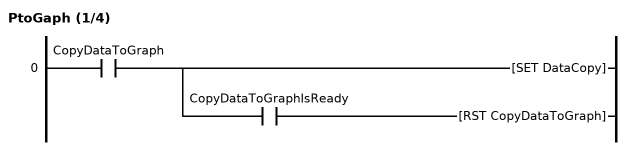
[picture p24: ladder of PtoGaph, rungs at steps 0 to 0]
0     LD      CopyDataToGraph
      SET     DataCopy
      AND     CopyDataToGraphIsReady
      RST     CopyDataToGraph
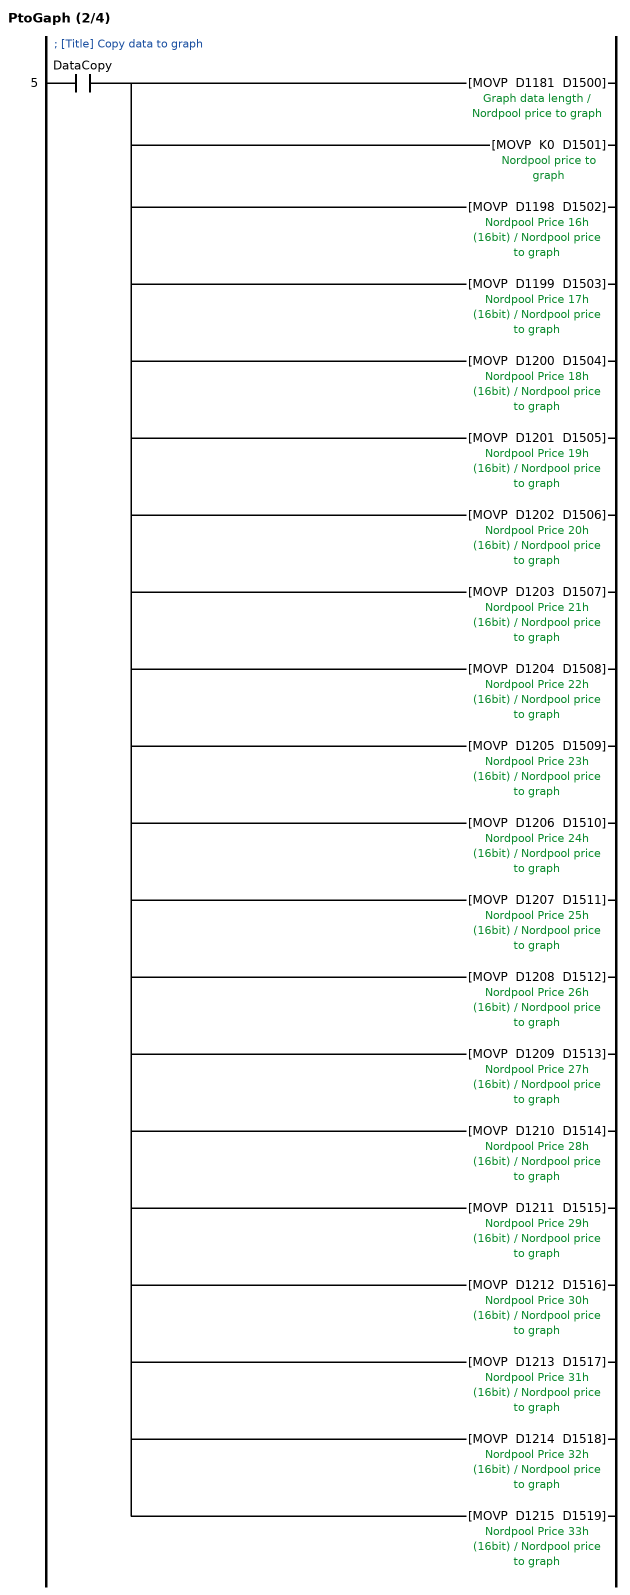
; [Title] Copy data to graph
5     LD      DataCopy
      MOVP    D1181 D1500  ; Graph data length / Nordpool price to graph
      MOVP    K0 D1501  ; Nordpool price to graph
      MOVP    D1198 D1502  ; Nordpool Price 16h (16bit) / Nordpool price to graph
      MOVP    D1199 D1503  ; Nordpool Price 17h (16bit) / Nordpool price to graph
      MOVP    D1200 D1504  ; Nordpool Price 18h (16bit) / Nordpool price to graph
      MOVP    D1201 D1505  ; Nordpool Price 19h (16bit) / Nordpool price to graph
      MOVP    D1202 D1506  ; Nordpool Price 20h (16bit) / Nordpool price to graph
      MOVP    D1203 D1507  ; Nordpool Price 21h (16bit) / Nordpool price to graph
      MOVP    D1204 D1508  ; Nordpool Price 22h (16bit) / Nordpool price to graph
      MOVP    D1205 D1509  ; Nordpool Price 23h (16bit) / Nordpool price to graph
      MOVP    D1206 D1510  ; Nordpool Price 24h (16bit) / Nordpool price to graph
      MOVP    D1207 D1511  ; Nordpool Price 25h (16bit) / Nordpool price to graph
      MOVP    D1208 D1512  ; Nordpool Price 26h (16bit) / Nordpool price to graph
      MOVP    D1209 D1513  ; Nordpool Price 27h (16bit) / Nordpool price to graph
      MOVP    D1210 D1514  ; Nordpool Price 28h (16bit) / Nordpool price to graph
      MOVP    D1211 D1515  ; Nordpool Price 29h (16bit) / Nordpool price to graph
      MOVP    D1212 D1516  ; Nordpool Price 30h (16bit) / Nordpool price to graph
      MOVP    D1213 D1517  ; Nordpool Price 31h (16bit) / Nordpool price to graph
      MOVP    D1214 D1518  ; Nordpool Price 32h (16bit) / Nordpool price to graph
      MOVP    D1215 D1519  ; Nordpool Price 33h (16bit) / Nordpool price to graph
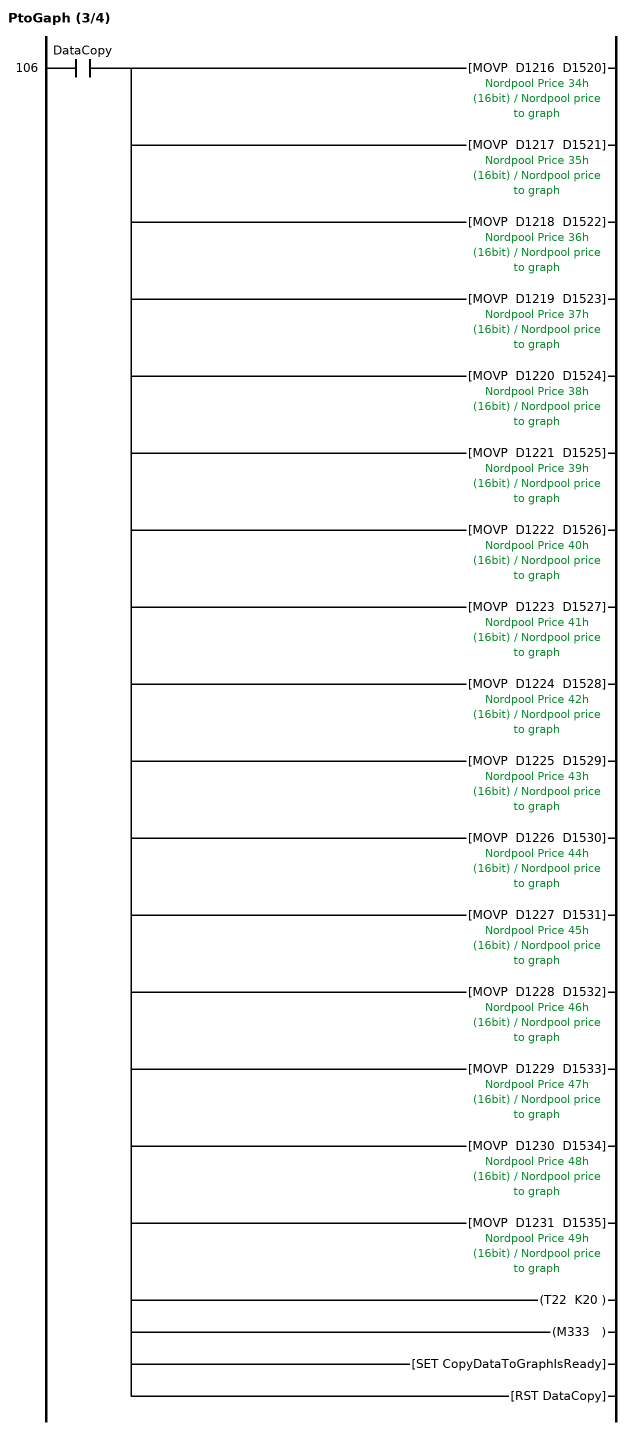
106   LD      DataCopy
      MOVP    D1216 D1520  ; Nordpool Price 34h (16bit) / Nordpool price to graph
      MOVP    D1217 D1521  ; Nordpool Price 35h (16bit) / Nordpool price to graph
      MOVP    D1218 D1522  ; Nordpool Price 36h (16bit) / Nordpool price to graph
      MOVP    D1219 D1523  ; Nordpool Price 37h (16bit) / Nordpool price to graph
      MOVP    D1220 D1524  ; Nordpool Price 38h (16bit) / Nordpool price to graph
      MOVP    D1221 D1525  ; Nordpool Price 39h (16bit) / Nordpool price to graph
      MOVP    D1222 D1526  ; Nordpool Price 40h (16bit) / Nordpool price to graph
      MOVP    D1223 D1527  ; Nordpool Price 41h (16bit) / Nordpool price to graph
      MOVP    D1224 D1528  ; Nordpool Price 42h (16bit) / Nordpool price to graph
      MOVP    D1225 D1529  ; Nordpool Price 43h (16bit) / Nordpool price to graph
      MOVP    D1226 D1530  ; Nordpool Price 44h (16bit) / Nordpool price to graph
      MOVP    D1227 D1531  ; Nordpool Price 45h (16bit) / Nordpool price to graph
      MOVP    D1228 D1532  ; Nordpool Price 46h (16bit) / Nordpool price to graph
      MOVP    D1229 D1533  ; Nordpool Price 47h (16bit) / Nordpool price to graph
      MOVP    D1230 D1534  ; Nordpool Price 48h (16bit) / Nordpool price to graph
      MOVP    D1231 D1535  ; Nordpool Price 49h (16bit) / Nordpool price to graph
      OUT     T22 K20
      OUT     M333
      SET     CopyDataToGraphIsReady
      RST     DataCopy
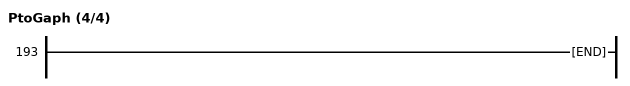
193   END
END_PROGRAM

PROGRAM SortData
VAR
  ValuesToSort1 : COUNTER;  (* Values to sorting *)
  Sortloop : DINT;  (* Sortng loop *)
  sortedelements : DINT;  (* sorted elements *)
  sortcycles : DINT;  (* Sorted cycles *)
  DataFucBlock : INT;  (* data sort counter *)
END_VAR
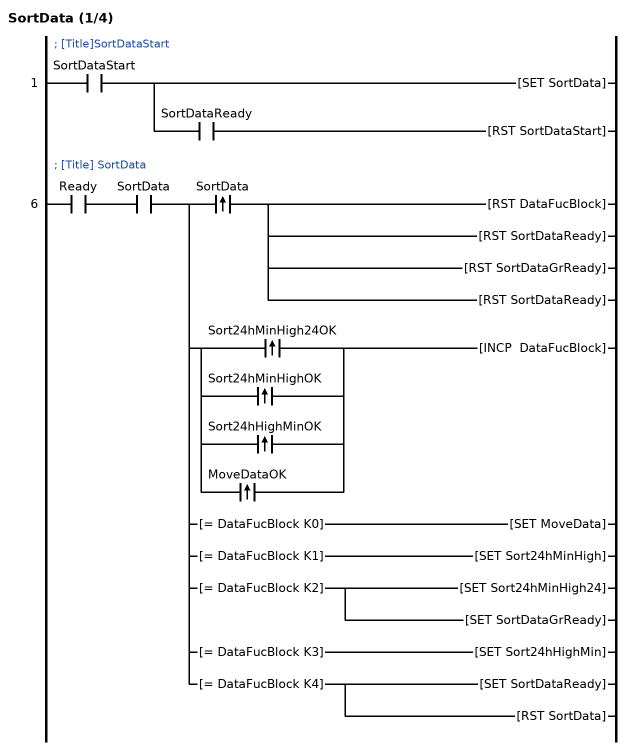
; [Title]SortDataStart
1     LD      SortDataStart
      SET     SortData
      AND     SortDataReady
      RST     SortDataStart
; [Title] SortData
6     LD      Ready
      AND     SortData
      MPS
      ANDP    SortData
      RST     DataFucBlock
      RST     SortDataReady
      RST     SortDataGrReady
      RST     SortDataReady
      MRD
      LDP     Sort24hMinHigh24OK
      ORP     Sort24hMinHighOK
      ORP     Sort24hHighMinOK
      ORP     MoveDataOK
      ANB
      INCP    DataFucBlock
      MRD
      AND=    DataFucBlock K0
      SET     MoveData
      MRD
      AND=    DataFucBlock K1
      SET     Sort24hMinHigh
      MRD
      AND=    DataFucBlock K2
      SET     Sort24hMinHigh24
      SET     SortDataGrReady
      MRD
      AND=    DataFucBlock K3
      SET     Sort24hHighMin
      MPP
      AND=    DataFucBlock K4
      SET     SortDataReady
      RST     SortData
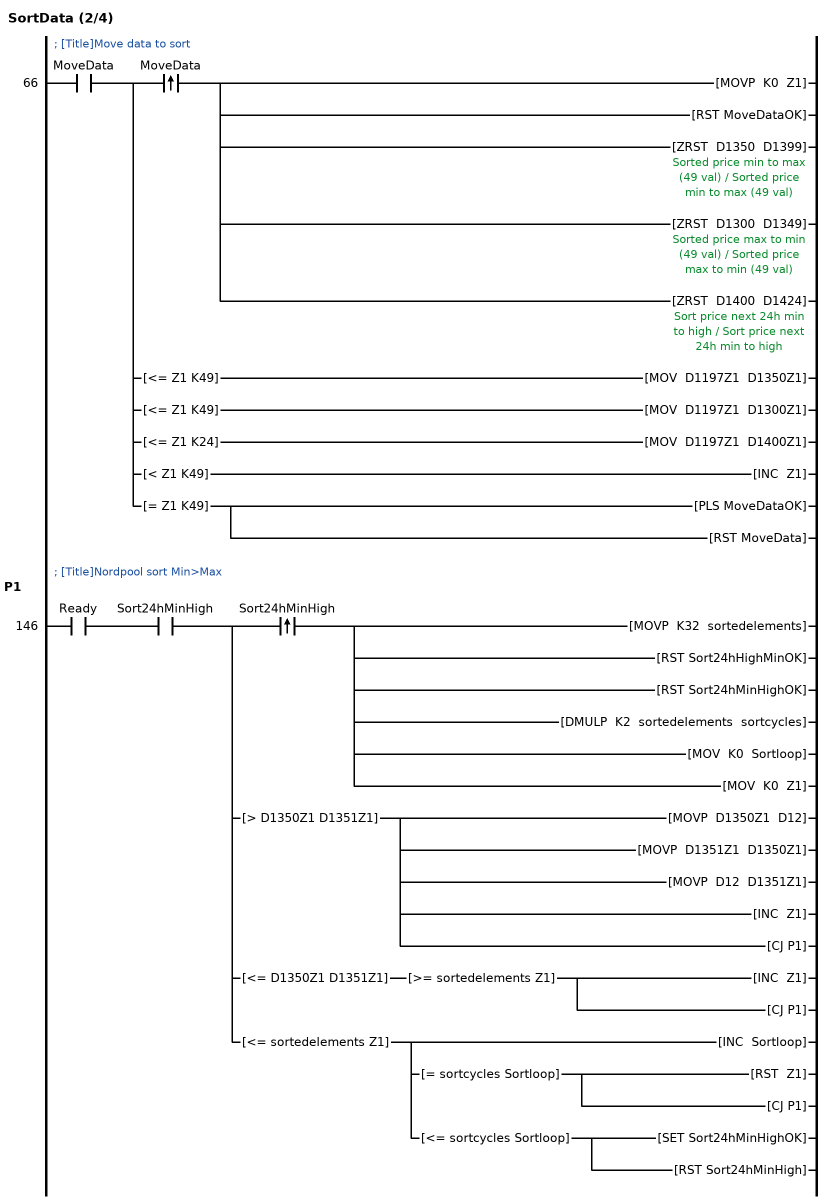
; [Title]Move data to sort
66    LD      MoveData
      MPS
      ANDP    MoveData
      MOVP    K0 Z1
      RST     MoveDataOK
      ZRST    D1350 D1399  ; Sorted price min to max (49 val) / Sorted price min to max (49 val)
        [note] Nordpool price min>max
      ZRST    D1300 D1349  ; Sorted price max to min (49 val) / Sorted price max to min (49 val)
        [note] ;Nordpool price max>min
      ZRST    D1400 D1424  ; Sort price next 24h min to high / Sort price next 24h min to high
        [note] ;Nordpool price 24h >max
      MRD
      AND<=   Z1 K49
      MOV     D1197Z1 D1350Z1
      MRD
      AND<=   Z1 K49
      MOV     D1197Z1 D1300Z1
      MRD
      AND<=   Z1 K24
      MOV     D1197Z1 D1400Z1
      MRD
      AND<    Z1 K49
      INC     Z1
      MPP
      AND=    Z1 K49
      PLS     MoveDataOK
      RST     MoveData
; [Title]Nordpool sort Min>Max
      P1
146   LD      Ready
      AND     Sort24hMinHigh
      MPS
      ANDP    Sort24hMinHigh
      MOVP    K32 sortedelements
      RST     Sort24hHighMinOK
      RST     Sort24hMinHighOK
      DMULP   K2 sortedelements sortcycles
      MOV     K0 Sortloop
      MOV     K0 Z1
      MRD
      AND>    D1350Z1 D1351Z1
      MOVP    D1350Z1 D12
      MOVP    D1351Z1 D1350Z1
      MOVP    D12 D1351Z1
      INC     Z1
      CJ      P1
      MRD
      AND<=   D1350Z1 D1351Z1
      AND>=   sortedelements Z1
      INC     Z1
      CJ      P1
      MPP
      AND<=   sortedelements Z1
      INC     Sortloop
      MPS
      AND=    sortcycles Sortloop
      RST     Z1
      CJ      P1
      MPP
      AND<=   sortcycles Sortloop
      SET     Sort24hMinHighOK
      RST     Sort24hMinHigh
; [Title]Nordpool sort Max>Min
      P2
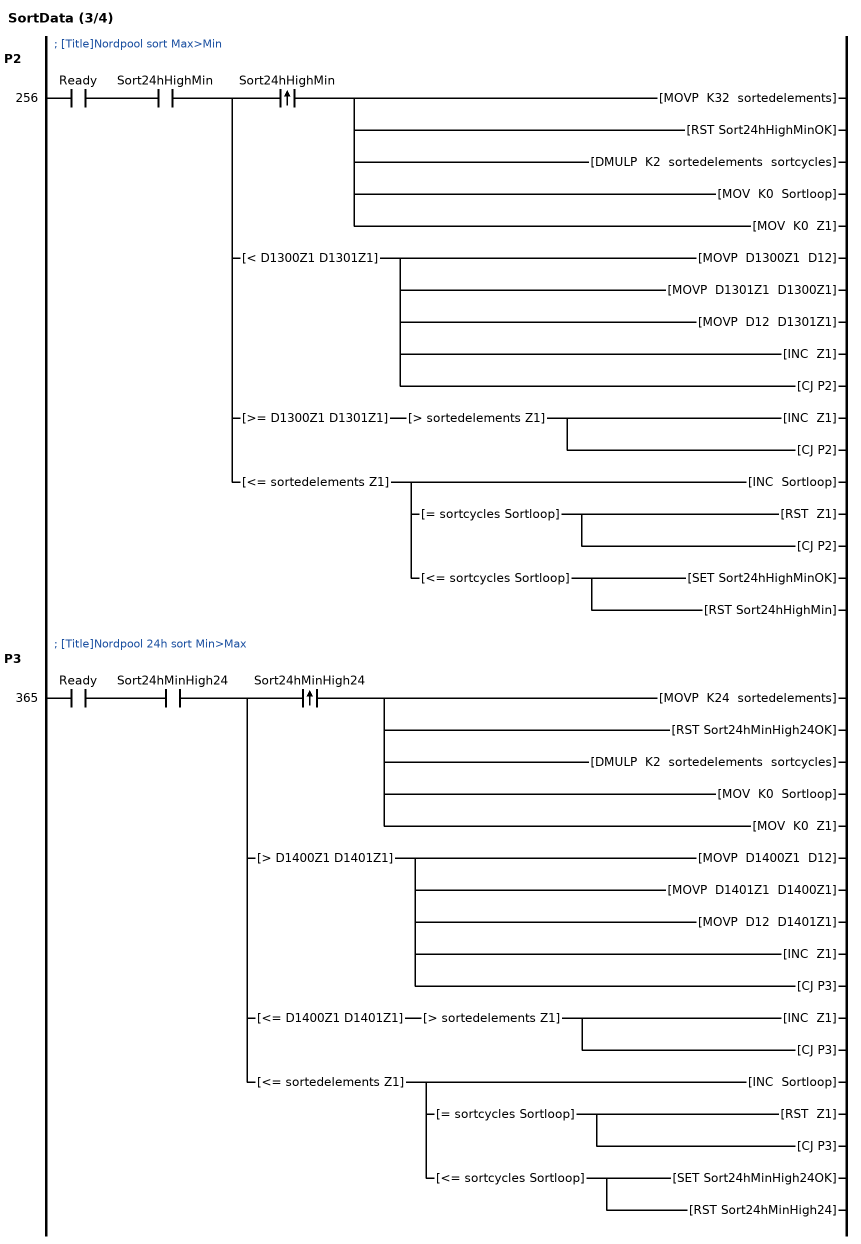
256   LD      Ready
      AND     Sort24hHighMin
      MPS
      ANDP    Sort24hHighMin
      MOVP    K32 sortedelements
      RST     Sort24hHighMinOK
      DMULP   K2 sortedelements sortcycles
      MOV     K0 Sortloop
      MOV     K0 Z1
      MRD
      AND<    D1300Z1 D1301Z1
      MOVP    D1300Z1 D12
      MOVP    D1301Z1 D1300Z1
      MOVP    D12 D1301Z1
      INC     Z1
      CJ      P2
      MRD
      AND>=   D1300Z1 D1301Z1
      AND>    sortedelements Z1
      INC     Z1
      CJ      P2
      MPP
      AND<=   sortedelements Z1
      INC     Sortloop
      MPS
      AND=    sortcycles Sortloop
      RST     Z1
      CJ      P2
      MPP
      AND<=   sortcycles Sortloop
      SET     Sort24hHighMinOK
      RST     Sort24hHighMin
; [Title]Nordpool 24h sort Min>Max
      P3
365   LD      Ready
      AND     Sort24hMinHigh24
      MPS
      ANDP    Sort24hMinHigh24
      MOVP    K24 sortedelements
      RST     Sort24hMinHigh24OK
      DMULP   K2 sortedelements sortcycles
      MOV     K0 Sortloop
      MOV     K0 Z1
      MRD
      AND>    D1400Z1 D1401Z1
      MOVP    D1400Z1 D12
      MOVP    D1401Z1 D1400Z1
      MOVP    D12 D1401Z1
      INC     Z1
      CJ      P3
      MRD
      AND<=   D1400Z1 D1401Z1
      AND>    sortedelements Z1
      INC     Z1
      CJ      P3
      MPP
      AND<=   sortedelements Z1
      INC     Sortloop
      MPS
      AND=    sortcycles Sortloop
      RST     Z1
      CJ      P3
      MPP
      AND<=   sortcycles Sortloop
      SET     Sort24hMinHigh24OK
      RST     Sort24hMinHigh24
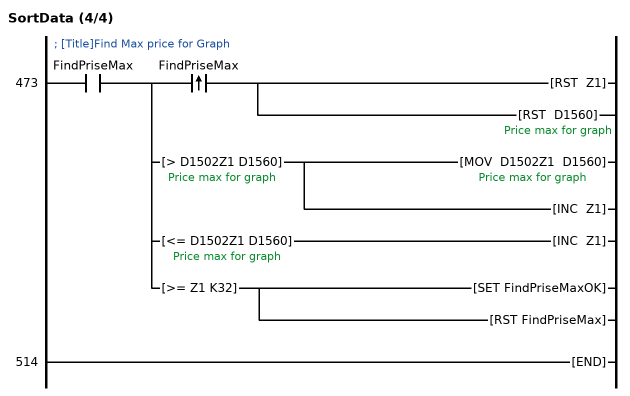
; [Title]Find Max price for Graph
473   LD      FindPriseMax
      MPS
      ANDP    FindPriseMax
      RST     Z1
      RST     D1560  ; Price max for graph
      MRD
      AND>    D1502Z1 D1560  ; Price max for graph
      MOV     D1502Z1 D1560
      INC     Z1
      MRD
      AND<=   D1502Z1 D1560  ; Price max for graph
      INC     Z1
      MPP
      AND>=   Z1 K32
      SET     FindPriseMaxOK
      RST     FindPriseMax
514   END
END_PROGRAM

PROGRAM WeathIN
VAR
  WeatherToGraph : BOOL;  (* Start wether data copy *)
  WeatherToGraphReady : BOOL;  (* Weather data is ready *)
  SumOfTemp : INT;  (* Sum of temp 24h *)
  SumOfWind : INT;  (* Sum of Wind 24h *)
  SumOfCloudy : INT;  (* Sum of clody 3h *)
END_VAR
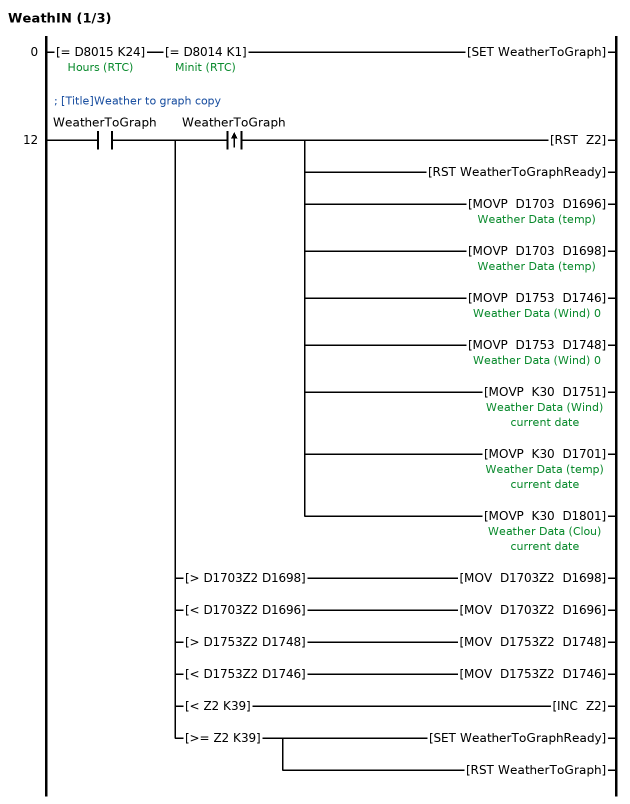
0     LD=     D8015 K24  ; Hours (RTC)
      AND=    D8014 K1  ; Minit (RTC)
      SET     WeatherToGraph
; [Title]Weather to graph copy
12    LD      WeatherToGraph
      MPS
      ANDP    WeatherToGraph
      RST     Z2
      RST     WeatherToGraphReady
      MOVP    D1703 D1696  ; Weather Data (temp)
      MOVP    D1703 D1698
      MOVP    D1753 D1746  ; Weather Data (Wind) 0
      MOVP    D1753 D1748
      MOVP    K30 D1751  ; Weather Data (Wind) current date
      MOVP    K30 D1701  ; Weather Data (temp) current date
      MOVP    K30 D1801  ; Weather Data (Clou) current date
      MRD
      AND>    D1703Z2 D1698
      MOV     D1703Z2 D1698
        [note] max temp for graphig ax
      MRD
      AND<    D1703Z2 D1696
      MOV     D1703Z2 D1696
        [note] min temp for garph ax
      MRD
      AND>    D1753Z2 D1748
      MOV     D1753Z2 D1748
        [note] max Wind for graphix ax
      MRD
      AND<    D1753Z2 D1746
      MOV     D1753Z2 D1746
        [note] min Wind for graphig ax
      MRD
      AND<    Z2 K39
      INC     Z2
      MPP
      AND>=   Z2 K39
      SET     WeatherToGraphReady
      RST     WeatherToGraph
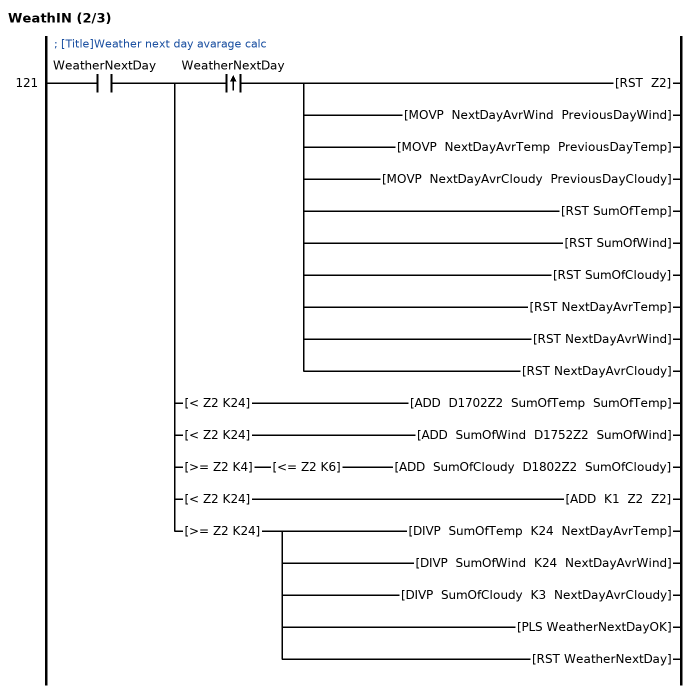
; [Title]Weather next day avarage calc
121   LD      WeatherNextDay
      MPS
      ANDP    WeatherNextDay
      RST     Z2
      MOVP    NextDayAvrWind PreviousDayWind
        [note] Data movement for previous day
      MOVP    NextDayAvrTemp PreviousDayTemp
      MOVP    NextDayAvrCloudy PreviousDayCloudy
      RST     SumOfTemp
      RST     SumOfWind
      RST     SumOfCloudy
      RST     NextDayAvrTemp
      RST     NextDayAvrWind
      RST     NextDayAvrCloudy
      MRD
      AND<    Z2 K24
      ADD     D1702Z2 SumOfTemp SumOfTemp
        [note] Data to average val.
      MRD
      AND<    Z2 K24
      ADD     SumOfWind D1752Z2 SumOfWind
      MRD
      AND>=   Z2 K4
      AND<=   Z2 K6
      ADD     SumOfCloudy D1802Z2 SumOfCloudy
      MRD
      AND<    Z2 K24
      ADD     K1 Z2 Z2
      MPP
      AND>=   Z2 K24
      DIVP    SumOfTemp K24 NextDayAvrTemp
        [note] Next day average prognosis
      DIVP    SumOfWind K24 NextDayAvrWind
      DIVP    SumOfCloudy K3 NextDayAvrCloudy
      PLS     WeatherNextDayOK
      RST     WeatherNextDay
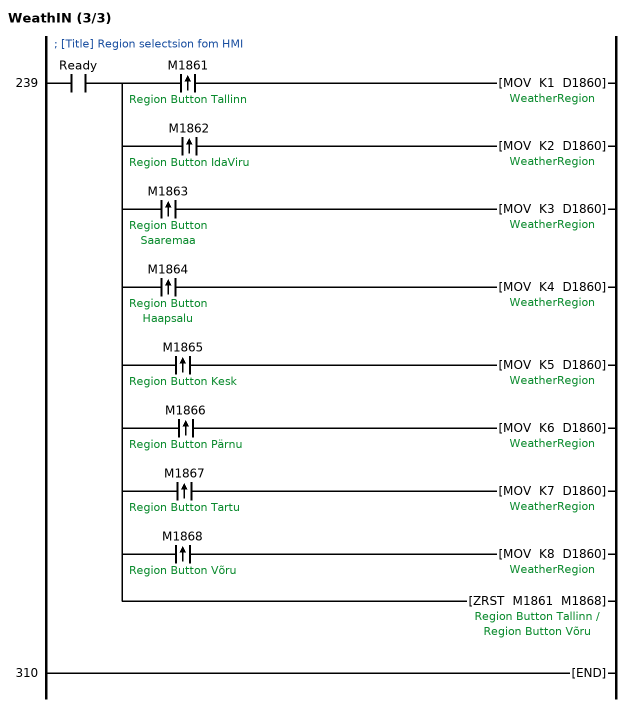
; [Title] Region selectsion fom HMI
239   LD      Ready
      MPS
      ANDP    M1861  ; Region Button Tallinn
      MOV     K1 D1860  ; WeatherRegion
      MRD
      ANDP    M1862  ; Region Button IdaViru
      MOV     K2 D1860
      MRD
      ANDP    M1863  ; Region Button Saaremaa
      MOV     K3 D1860
      MRD
      ANDP    M1864  ; Region Button Haapsalu
      MOV     K4 D1860
      MRD
      ANDP    M1865  ; Region Button Kesk
      MOV     K5 D1860
      MRD
      ANDP    M1866  ; Region Button Pärnu
      MOV     K6 D1860
      MRD
      ANDP    M1867  ; Region Button Tartu
      MOV     K7 D1860
      MRD
      ANDP    M1868  ; Region Button Võru
      MOV     K8 D1860
      MPP
      ZRST    M1861 M1868
310   END
END_PROGRAM

PROGRAM Energy
VAR
  TableColumnDIV : DINT;  (* Table column division *)
  TableRowDIV : DINT;  (* Find table data row *)
  DataInTableColumn : DINT;  (* Radiatsion in teable column *)
  WriteEnergyDataRequirement : INT;  (* Energy data for data table *)
  TankTempSum : DINT;  (* Tank temp low and high temp sum. *)
  TankTempAvr : DINT;  (* Tank temp average temp *)
  TankTempLiter : DINT;  (* Tank temp * liter *)
  TankEnergyCapacity : DINT;  (* Tank  energy capacity cap. wh*100 *)
  test : BOOL;  (* Test Flag *)
  test2 : BOOL;  (* test2 *)
  HeatInLastMinit : DINT;  (* Heat in last minit *)
  CountedHours : INT;  (* Number of hours counted *)
  FullDay : BOOL;  (* Full the day is counted *)
  EndHours : INT;  (* first minute counter *)
  EnergyConsumptionYesterdayPerM2 : DINT;  (* Energy consumption last day value per m2 *)
  SolarRadiation_x_Cludy : DINT;  (* Solar radiation max x cloudy % *)
  TemperatureDifference : INT;  (* Temperature difference (20C - previous day prognose) *)
  RadiationWeatherCalc : BOOL;  (* Radiation and weather Calc for table *)
END_VAR
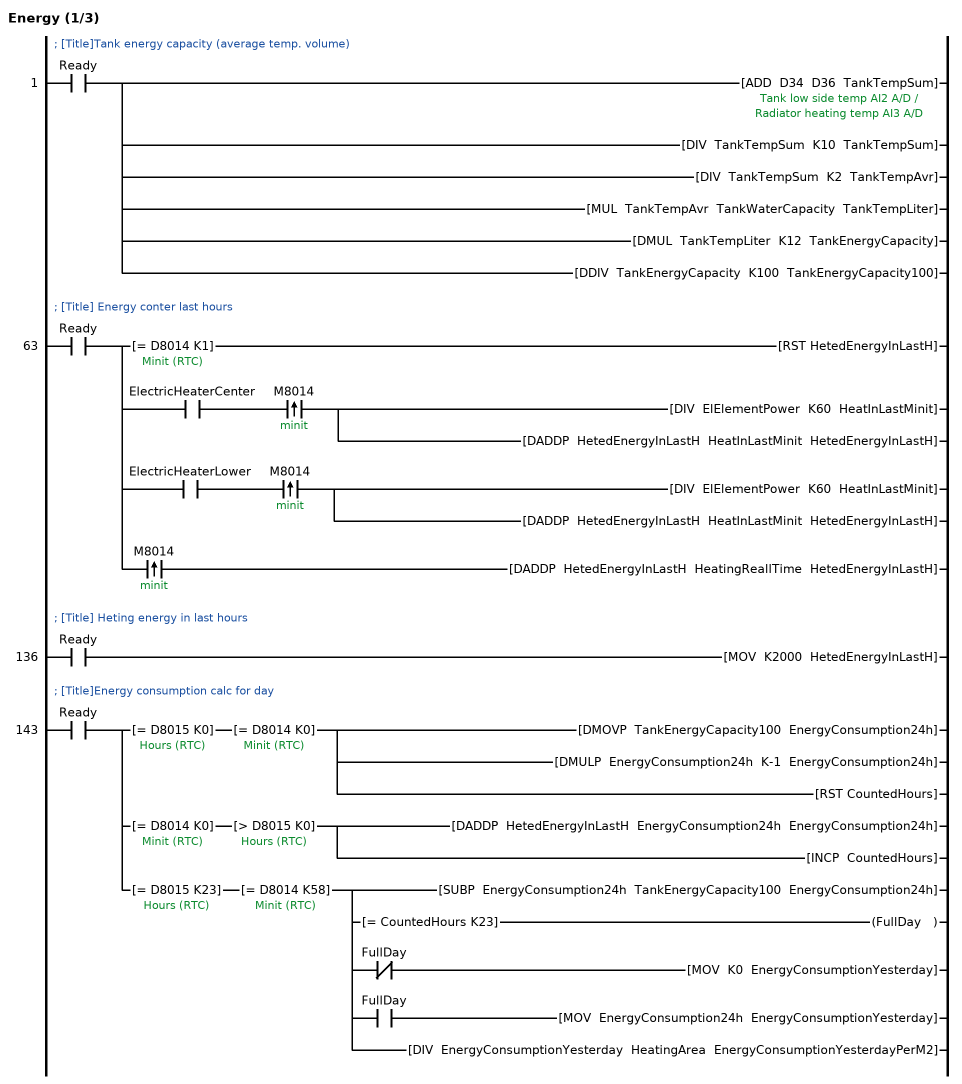
; [Title]Tank energy capacity (average temp. volume)
1     LD      Ready
      ADD     D34 D36 TankTempSum  ; Tank low side temp AI2 A/D / Radiator heating temp AI3 A/D
        [note] Average temp
      DIV     TankTempSum K10 TankTempSum
        [note] To temp (C)
      DIV     TankTempSum K2 TankTempAvr
        [note] avr temp
      MUL     TankTempAvr TankWaterCapacity TankTempLiter
        [note] calc temp*volume
      DMUL    TankTempLiter K12 TankEnergyCapacity
        [note] (temp*liter) x energy capacity
      DDIV    TankEnergyCapacity K100 TankEnergyCapacity100
        [note] reduction wh
; [Title] Energy conter last hours
63    LD      Ready
      MPS
      AND=    D8014 K1  ; Minit (RTC)
      RST     HetedEnergyInLastH
      MRD
      AND     ElectricHeaterCenter
      ANDP    M8014  ; minit
      DIV     ElElementPower K60 HeatInLastMinit
      DADDP   HetedEnergyInLastH HeatInLastMinit HetedEnergyInLastH
      MRD
      AND     ElectricHeaterLower
      ANDP    M8014  ; minit
      DIV     ElElementPower K60 HeatInLastMinit
      DADDP   HetedEnergyInLastH HeatInLastMinit HetedEnergyInLastH
      MPP
      ANDP    M8014  ; minit
      DADDP   HetedEnergyInLastH HeatingReallTime HetedEnergyInLastH
; [Title] Heting energy in last hours
136   LD      Ready
      MOV     K2000 HetedEnergyInLastH
; [Title]Energy consumption calc for day
143   LD      Ready
      MPS
      AND=    D8015 K0  ; Hours (RTC)
      AND=    D8014 K0  ; Minit (RTC)
      DMOVP   TankEnergyCapacity100 EnergyConsumption24h
        [note] amount of energy
      DMULP   EnergyConsumption24h K-1 EnergyConsumption24h
        [note] negative initial value
      RST     CountedHours
      MRD
      AND=    D8014 K0  ; Minit (RTC)
      AND>    D8015 K0  ; Hours (RTC)
      DADDP   HetedEnergyInLastH EnergyConsumption24h EnergyConsumption24h
        [note] energy added every hours
      INCP    CountedHours
        [note] added hours counter
      MPP
      AND=    D8015 K23  ; Hours (RTC)
      AND=    D8014 K58  ; Minit (RTC)
      SUBP    EnergyConsumption24h TankEnergyCapacity100 EnergyConsumption24h
        [note] energy to end the day
      MPS
      AND=    CountedHours K23
      OUT     FullDay
      MRD
      ANI     FullDay
      MOV     K0 EnergyConsumptionYesterday
        [note] if not full day then energy 0
      MRD
      AND     FullDay
      MOV     EnergyConsumption24h EnergyConsumptionYesterday
        [note] energy consumed per day
      MPP
      DIV     EnergyConsumptionYesterday HeatingArea EnergyConsumptionYesterdayPerM2
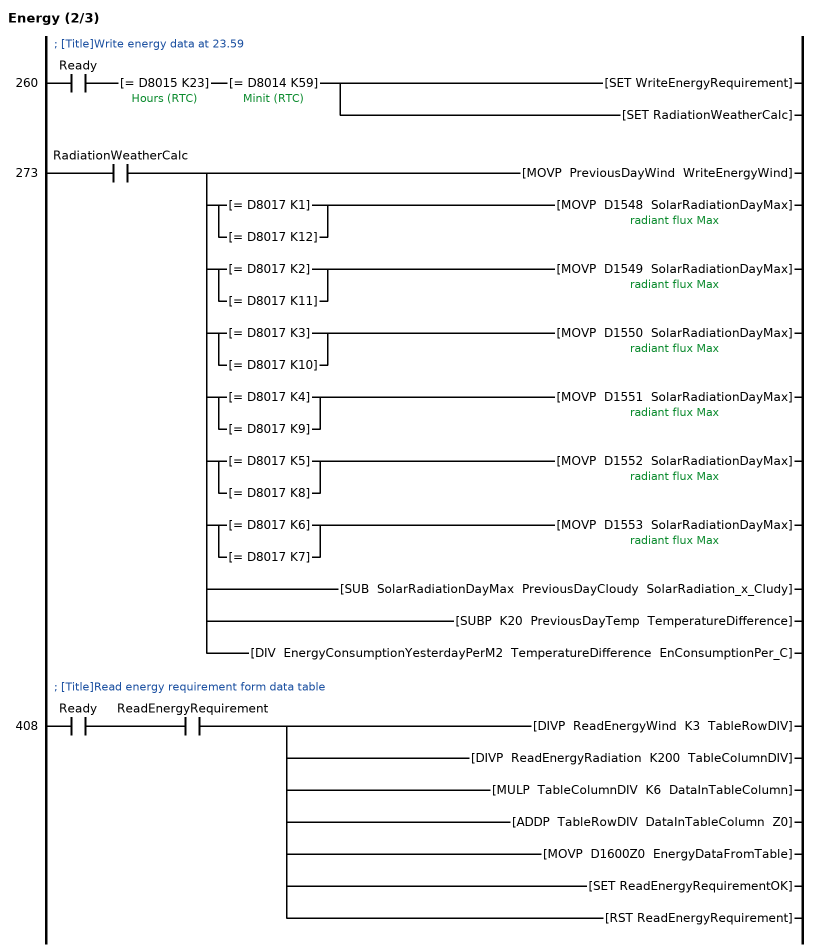
; [Title]Write energy data at 23.59
260   LD      Ready
      AND=    D8015 K23  ; Hours (RTC)
      AND=    D8014 K59  ; Minit (RTC)
      SET     WriteEnergyRequirement
      SET     RadiationWeatherCalc
273   LD      RadiationWeatherCalc
      MOVP    PreviousDayWind WriteEnergyWind
      MPS
      LD=     D8017 K1
      OR=     D8017 K12
      ANB
      MOVP    D1548 SolarRadiationDayMax  ; radiant flux Max
        [note] Solar radiation per month
      MRD
      LD=     D8017 K2
      OR=     D8017 K11
      ANB
      MOVP    D1549 SolarRadiationDayMax  ; radiant flux Max
      MRD
      LD=     D8017 K3
      OR=     D8017 K10
      ANB
      MOVP    D1550 SolarRadiationDayMax  ; radiant flux Max
      MRD
      LD=     D8017 K4
      OR=     D8017 K9
      ANB
      MOVP    D1551 SolarRadiationDayMax  ; radiant flux Max
      MRD
      LD=     D8017 K5
      OR=     D8017 K8
      ANB
      MOVP    D1552 SolarRadiationDayMax  ; radiant flux Max
      MRD
      LD=     D8017 K6
      OR=     D8017 K7
      ANB
      MOVP    D1553 SolarRadiationDayMax  ; radiant flux Max
      MPP
      SUB     SolarRadiationDayMax PreviousDayCloudy SolarRadiation_x_Cludy
        [note] Max energy x cloudy %
      SUBP    K20 PreviousDayTemp TemperatureDifference
        [note] Temp differents (20C - prognose)
      DIV     EnergyConsumptionYesterdayPerM2 TemperatureDifference EnConsumptionPer_C
        [note] energy consumption per degree
; [Title]Read energy requirement form data table
408   LD      Ready
      AND     ReadEnergyRequirement
      DIVP    ReadEnergyWind K3 TableRowDIV
      DIVP    ReadEnergyRadiation K200 TableColumnDIV
      MULP    TableColumnDIV K6 DataInTableColumn
      ADDP    TableRowDIV DataInTableColumn Z0
      MOVP    D1600Z0 EnergyDataFromTable
      SET     ReadEnergyRequirementOK
      RST     ReadEnergyRequirement
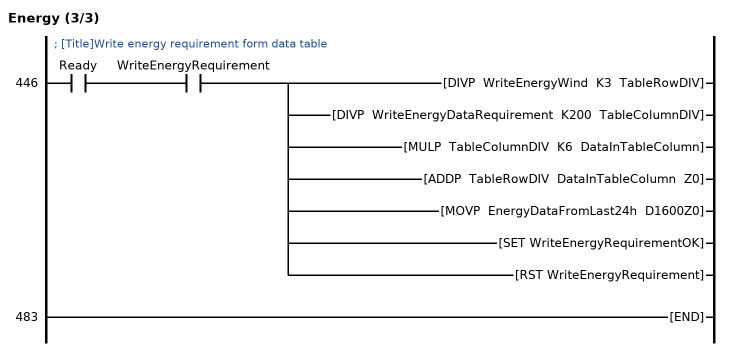
; [Title]Write energy requirement form data table
446   LD      Ready
      AND     WriteEnergyRequirement
      DIVP    WriteEnergyWind K3 TableRowDIV
      DIVP    WriteEnergyDataRequirement K200 TableColumnDIV
      MULP    TableColumnDIV K6 DataInTableColumn
      ADDP    TableRowDIV DataInTableColumn Z0
      MOVP    EnergyDataFromLast24h D1600Z0
      SET     WriteEnergyRequirementOK
      RST     WriteEnergyRequirement
483   END
END_PROGRAM

PROGRAM IO_CONF
VAR
  FlowPulse : INT;  (* Flow sensor pulse input *)
  FlowPulseInMinit : INT;  (* Flow pulses per minit *)
  HeatFlowLitersDay : INT;  (* Heat flow liter in Day *)
  test : BOOL;
  HeatingTempDiffrents : INT;  (* Heating temp differents (heat-return water) *)
  HeatWaterPoewer : DINT;  (* Heat water energy *)
END_VAR
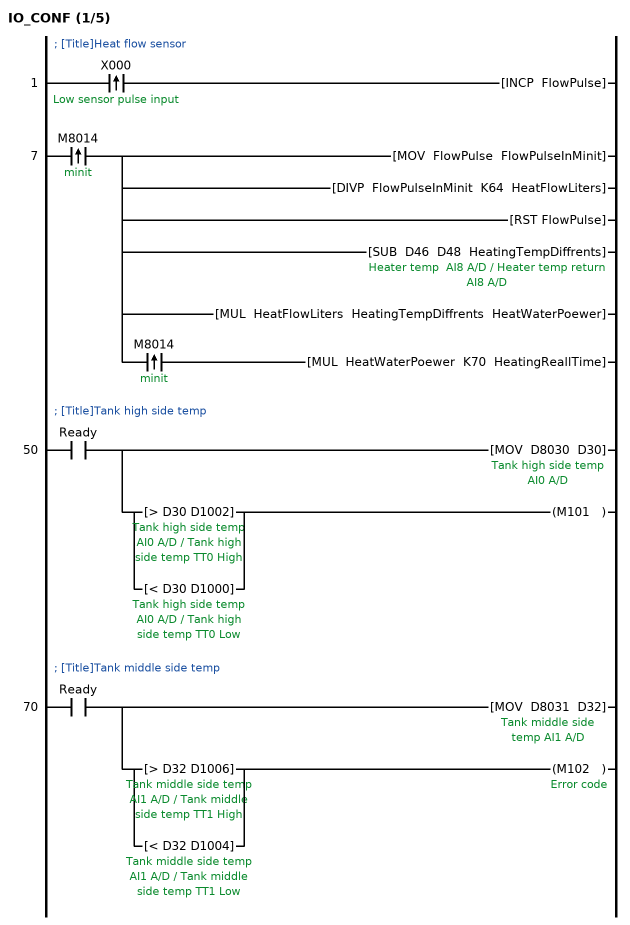
; [Title]Heat flow sensor
1     LDP     X000  ; Low sensor pulse input
      INCP    FlowPulse
        [note] count pule
7     LDP     M8014  ; minit
      MOV     FlowPulse FlowPulseInMinit
        [note] Add data to minit register
      DIVP    FlowPulseInMinit K64 HeatFlowLiters
        [note] number conversion to l/min
      RST     FlowPulse
        [note] reset counter
      SUB     D46 D48 HeatingTempDiffrents  ; Heater temp  AI8 A/D / Heater temp return AI8 A/D
        [note] Hetin temp differents
      MUL     HeatFlowLiters HeatingTempDiffrents HeatWaterPoewer
      ANDP    M8014  ; minit
      MUL     HeatWaterPoewer K70 HeatingReallTime
; [Title]Tank high side temp
50    LD      Ready
      MOV     D8030 D30  ; Tank high side temp AI0 A/D
        [note] Tank high side temp TT0
      LD>     D30 D1002  ; Tank high side temp AI0 A/D / Tank high side temp TT0 High
      OR<     D30 D1000  ; Tank high side temp AI0 A/D / Tank high side temp TT0 Low
      ANB
      OUT     M101
; [Title]Tank middle side temp
70    LD      Ready
      MOV     D8031 D32  ; Tank middle side temp AI1 A/D
        [note] Tank middle side temp TT1
      LD>     D32 D1006  ; Tank middle side temp AI1 A/D / Tank middle side temp TT1 High
      OR<     D32 D1004  ; Tank middle side temp AI1 A/D / Tank middle side temp TT1 Low
      ANB
      OUT     M102  ; Error code
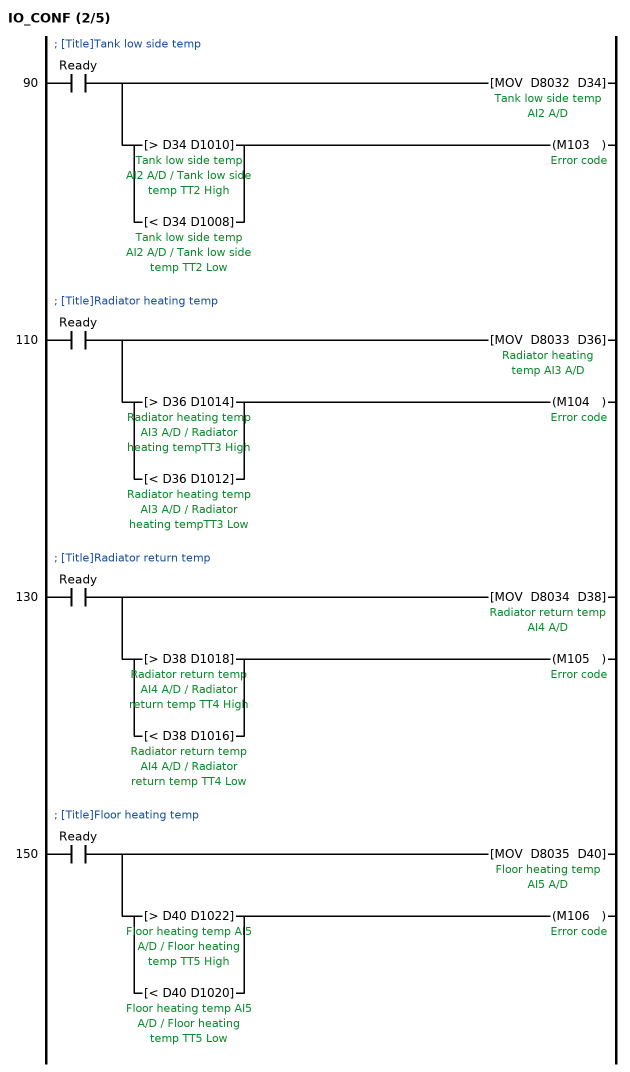
; [Title]Tank low side temp
90    LD      Ready
      MOV     D8032 D34  ; Tank low side temp AI2 A/D
        [note] Tank low side temp TT2
      LD>     D34 D1010  ; Tank low side temp AI2 A/D / Tank low side temp TT2 High
      OR<     D34 D1008  ; Tank low side temp AI2 A/D / Tank low side temp TT2 Low
      ANB
      OUT     M103  ; Error code
; [Title]Radiator heating temp
110   LD      Ready
      MOV     D8033 D36  ; Radiator heating temp AI3 A/D
        [note] Radiator heating tempTT3
      LD>     D36 D1014  ; Radiator heating temp AI3 A/D / Radiator heating tempTT3 High
      OR<     D36 D1012  ; Radiator heating temp AI3 A/D / Radiator heating tempTT3 Low
      ANB
      OUT     M104  ; Error code
; [Title]Radiator return temp
130   LD      Ready
      MOV     D8034 D38  ; Radiator return temp AI4 A/D
        [note] Radiator return temp TT4
      LD>     D38 D1018  ; Radiator return temp AI4 A/D / Radiator return temp TT4 High
      OR<     D38 D1016  ; Radiator return temp AI4 A/D / Radiator return temp TT4 Low
      ANB
      OUT     M105  ; Error code
; [Title]Floor heating temp
150   LD      Ready
      MOV     D8035 D40  ; Floor heating temp AI5 A/D
        [note] Floor heating temp TT5
      LD>     D40 D1022  ; Floor heating temp AI5 A/D / Floor heating temp TT5 High
      OR<     D40 D1020  ; Floor heating temp AI5 A/D / Floor heating temp TT5 Low
      ANB
      OUT     M106  ; Error code
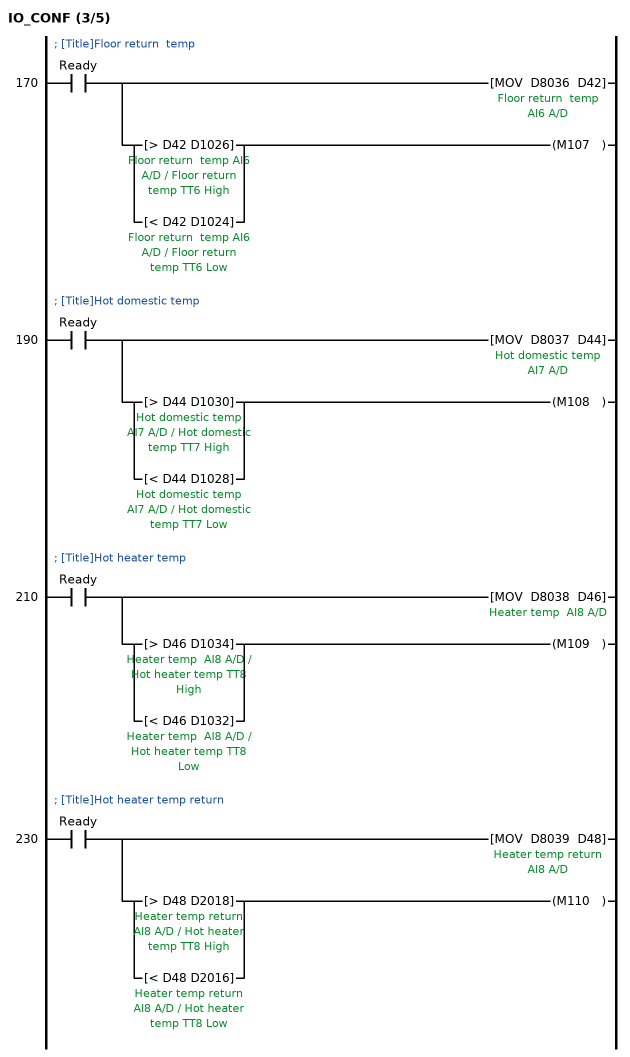
; [Title]Floor return  temp
170   LD      Ready
      MOV     D8036 D42  ; Floor return  temp AI6 A/D
        [note] Floor return  temp TT6
      LD>     D42 D1026  ; Floor return  temp AI6 A/D / Floor return  temp TT6 High
      OR<     D42 D1024  ; Floor return  temp AI6 A/D / Floor return  temp TT6 Low
      ANB
      OUT     M107
; [Title]Hot domestic temp
190   LD      Ready
      MOV     D8037 D44  ; Hot domestic temp AI7 A/D
        [note] Hot domestic temp TT7
      LD>     D44 D1030  ; Hot domestic temp AI7 A/D / Hot domestic temp TT7 High
      OR<     D44 D1028  ; Hot domestic temp AI7 A/D / Hot domestic temp TT7 Low
      ANB
      OUT     M108
; [Title]Hot heater temp
210   LD      Ready
      MOV     D8038 D46
        [note] Hot heater temp TT8
      LD>     D46 D1034  ; Heater temp  AI8 A/D / Hot heater temp TT8 High
      OR<     D46 D1032  ; Heater temp  AI8 A/D / Hot heater temp TT8 Low
      ANB
      OUT     M109
; [Title]Hot heater temp return
230   LD      Ready
      MOV     D8039 D48
        [note] Hot heater temp TT8
      LD>     D48 D2018  ; Heater temp return AI8 A/D / Hot heater temp TT8 High
      OR<     D48 D2016  ; Heater temp return AI8 A/D / Hot heater temp TT8 Low
      ANB
      OUT     M110
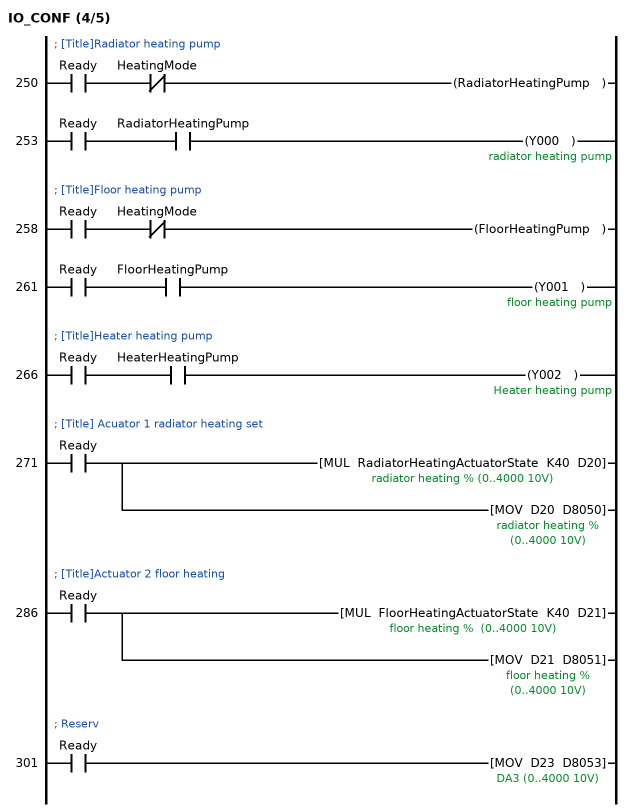
; [Title]Radiator heating pump
250   LD      Ready
      ANI     HeatingMode
      OUT     RadiatorHeatingPump
253   LD      Ready
      AND     RadiatorHeatingPump
      OUT     Y000  ; radiator heating pump
        [note] radiator heating pump
; [Title]Floor heating pump
258   LD      Ready
      ANI     HeatingMode
      OUT     FloorHeatingPump
261   LD      Ready
      AND     FloorHeatingPump
      OUT     Y001  ; floor heating pump
        [note] floor heating pump
; [Title]Heater heating pump
266   LD      Ready
      AND     HeaterHeatingPump
      OUT     Y002  ; Heater heating pump
        [note] Heater heating pump
; [Title] Acuator 1 radiator heating set
271   LD      Ready
      MUL     RadiatorHeatingActuatorState K40 D20  ; radiator heating % (0..4000 10V)
      MOV     D20 D8050
        [note] Acuator 1 radiator heating
; [Title]Actuator 2 floor heating
286   LD      Ready
      MUL     FloorHeatingActuatorState K40 D21  ; floor heating %  (0..4000 10V)
      MOV     D21 D8051
        [note] Actuator 2 floor heating
; Reserv
301   LD      Ready
      MOV     D23 D8053  ; DA3 (0..4000 10V)
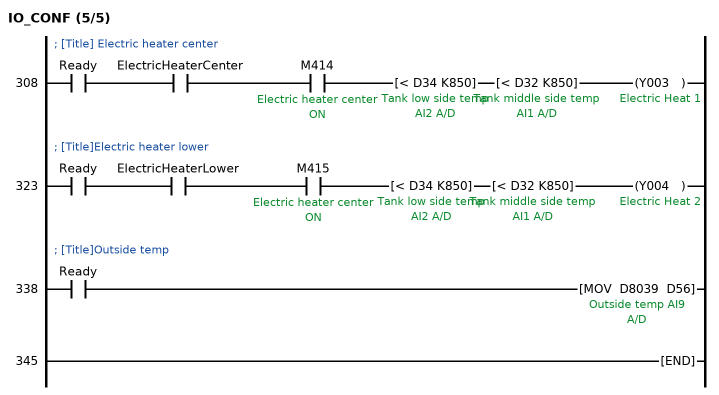
; [Title] Electric heater center
308   LD      Ready
      AND     ElectricHeaterCenter
      AND     M414  ; Electric heater center ON
      AND<    D34 K850  ; Tank low side temp AI2 A/D
      AND<    D32 K850  ; Tank middle side temp AI1 A/D
      OUT     Y003  ; Electric Heat 1
; [Title]Electric heater lower
323   LD      Ready
      AND     ElectricHeaterLower
      AND     M415  ; Electric heater center ON
      AND<    D34 K850  ; Tank low side temp AI2 A/D
      AND<    D32 K850  ; Tank middle side temp AI1 A/D
      OUT     Y004  ; Electric Heat 2
; [Title]Outside temp
338   LD      Ready
      MOV     D8039 D56  ; Outside temp AI9 A/D
        [note] Outside temp TT9
345   END
END_PROGRAM

PROGRAM Ring1_R
VAR
  TempShift : DINT;  (* Temerature sift for copensatsion *)
  Ring1ShiftAdd : DINT;  (* Temerature correctsion for Add *)
  Ring1ShiftAdded : DINT;  (* Target temp x 10 *)
  TempDiff : DINT;  (* Heat Graph temp difference *)
  TempDiffPer1C : DINT;  (* Temperature differens per 1c *)
  BaseTemp : INT;  (* Base temperatuere for calc *)
  OutOfTemp : BOOL;  (* Outside temp out of regutalatsion *)
  SetValue : INT;  (* Value from Graph *)
  TempdifferentsforPID : INT;  (* Temp different for PID *)
  TempInc : INT;  (* Temperature increment to actuator *)
  Ring1Interval : TIMER;  (* Ring 1 actuator valve update interval *)
  changeable : BOOL;  (* temperatuure need correctsion *)
  changeable2 : BOOL;
  TempdifferentsforPIDcor : DINT;  (* Corrected actuator value change *)
  Canadd : BOOL;  (* Can add more value *)
  CanTadd : BOOL;  (* Cant add more val *)
END_VAR
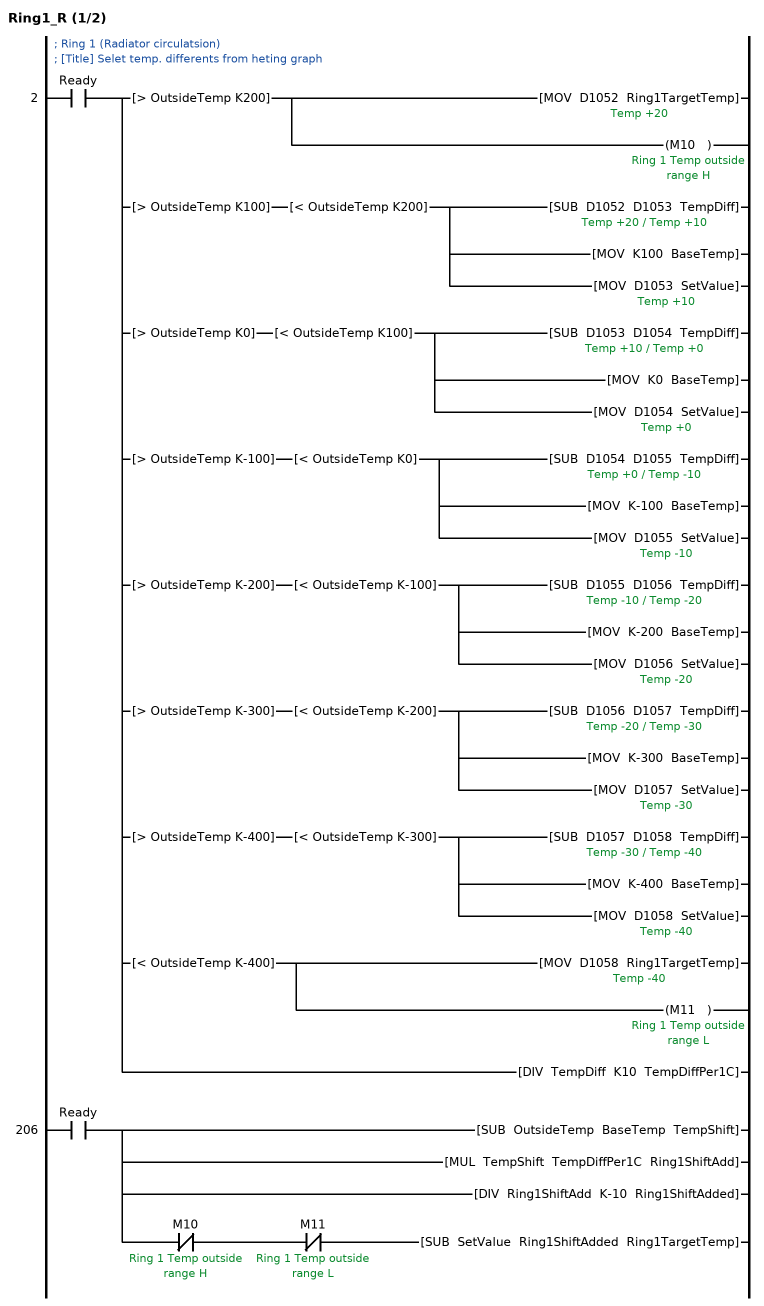
; Ring 1 (Radiator circulatsion)
; [Title] Selet temp. differents from heting graph
2     LD      Ready
      MPS
      AND>    OutsideTemp K200
      MOV     D1052 Ring1TargetTemp  ; Temp +20
        [note] Data from heating graph
      OUT     M10  ; Ring 1 Temp outside range H
      MRD
      AND>    OutsideTemp K100
      AND<    OutsideTemp K200
      SUB     D1052 D1053 TempDiff  ; Temp +10
      MOV     K100 BaseTemp
      MOV     D1053 SetValue
      MRD
      AND>    OutsideTemp K0
      AND<    OutsideTemp K100
      SUB     D1053 D1054 TempDiff  ; Temp +0
      MOV     K0 BaseTemp
      MOV     D1054 SetValue
      MRD
      AND>    OutsideTemp K-100
      AND<    OutsideTemp K0
      SUB     D1054 D1055 TempDiff  ; Temp -10
      MOV     K-100 BaseTemp
      MOV     D1055 SetValue
      MRD
      AND>    OutsideTemp K-200
      AND<    OutsideTemp K-100
      SUB     D1055 D1056 TempDiff  ; Temp -20
      MOV     K-200 BaseTemp
      MOV     D1056 SetValue
      MRD
      AND>    OutsideTemp K-300
      AND<    OutsideTemp K-200
      SUB     D1056 D1057 TempDiff  ; Temp -30
      MOV     K-300 BaseTemp
      MOV     D1057 SetValue
      MRD
      AND>    OutsideTemp K-400
      AND<    OutsideTemp K-300
      SUB     D1057 D1058 TempDiff  ; Temp -40
      MOV     K-400 BaseTemp
      MOV     D1058 SetValue
      MRD
      AND<    OutsideTemp K-400
      MOV     D1058 Ring1TargetTemp
        [note] Data from heating graph
      OUT     M11  ; Ring 1 Temp outside range L
      MPP
      DIV     TempDiff K10 TempDiffPer1C
        [note] Calculated differents per 1C
206   LD      Ready
      SUB     OutsideTemp BaseTemp TempShift
        [note] Temp differents
      MUL     TempShift TempDiffPer1C Ring1ShiftAdd
        [note] Temp diffrents  per 1C
      DIV     Ring1ShiftAdd K-10 Ring1ShiftAdded
      ANI     M10  ; Ring 1 Temp outside range H
      ANI     M11  ; Ring 1 Temp outside range L
      SUB     SetValue Ring1ShiftAdded Ring1TargetTemp
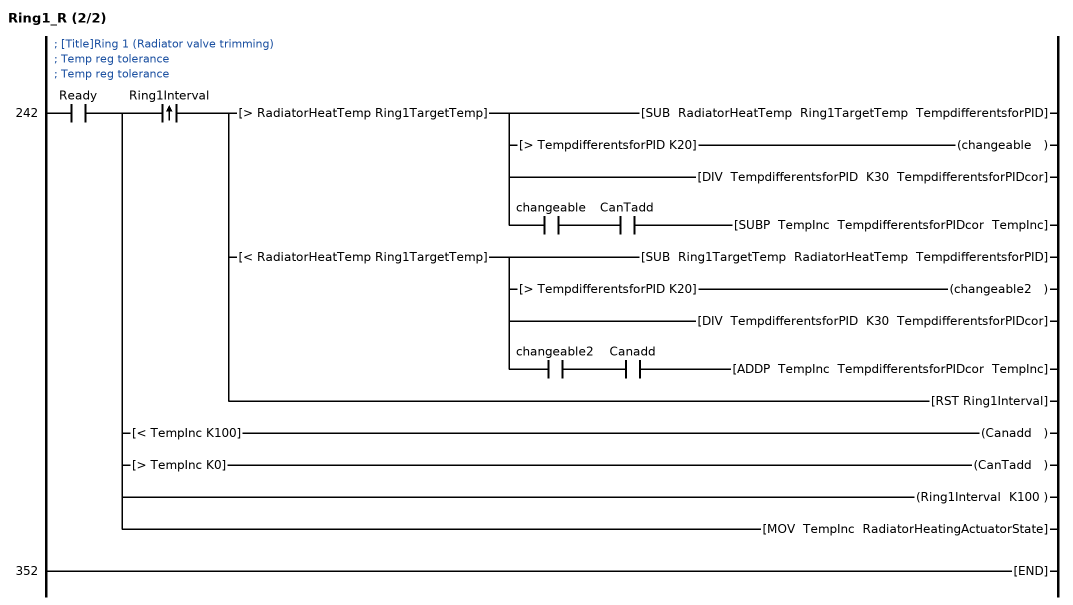
; [Title]Ring 1 (Radiator valve trimming)
; Temp reg tolerance
; Temp reg tolerance
242   LD      Ready
      MPS
      ANDP    Ring1Interval
      MPS
      AND>    RadiatorHeatTemp Ring1TargetTemp
      SUB     RadiatorHeatTemp Ring1TargetTemp TempdifferentsforPID
        [note] Calc temp differents for PID
      MPS
      AND>    TempdifferentsforPID K20
      OUT     changeable
        [note] Temp reg tolerance
      MPP
      DIV     TempdifferentsforPID K30 TempdifferentsforPIDcor
        [note] PID to actuator (%)
      AND     changeable
      AND     CanTadd
      SUBP    TempInc TempdifferentsforPIDcor TempInc
        [note] Correctsion actuator value (%)
      MRD
      AND<    RadiatorHeatTemp Ring1TargetTemp
      SUB     Ring1TargetTemp RadiatorHeatTemp TempdifferentsforPID
        [note] Calc temp differents for PID
      MPS
      AND>    TempdifferentsforPID K20
      OUT     changeable2
        [note] Temp reg tolerance
      MPP
      DIV     TempdifferentsforPID K30 TempdifferentsforPIDcor
        [note] PID to actuator (%)
      AND     changeable2
      AND     Canadd
      ADDP    TempInc TempdifferentsforPIDcor TempInc
        [note] Correctsion actuator value (%)
      MPP
      RST     Ring1Interval
      MRD
      AND<    TempInc K100
      OUT     Canadd
        [note] Actuator range control
      MRD
      AND>    TempInc K0
      OUT     CanTadd
      MPP
      OUT     Ring1Interval K100
      MOV     TempInc RadiatorHeatingActuatorState
352   END
END_PROGRAM

PROGRAM Ring2_F
VAR
  TempDiffPer1C : DINT;  (* Temerature differents pes 1 C *)
  TempShift : DINT;  (* Temperature shift *)
  Ring2ShiftAdd : DINT;
  Ring2ShiftAdded : DINT;
  TempDiff : DINT;  (* Heat Graph temp difference *)
  BaseTemp : INT;  (* Base temperatuere for calc *)
  SetValue : INT;  (* Value from Graph *)
  Ring2Interval : TIMER;  (* Ring 1 actuator valve update interval *)
  TempdifferentsforPID : INT;  (* Temp different for PID *)
  TempInc : INT;  (* Temperature increment to actuator *)
  Ring1Interval : TIMER;  (* Ring 1 actuator valve update interval *)
  changeable : BOOL;  (* temperatuure need correctsion *)
  TempdifferentsforPIDcor : DINT;  (* Corrected actuator value change *)
  Canadd : BOOL;  (* Can add more value *)
  CanTadd : BOOL;  (* Cant add more val *)
  changeable2 : BOOL;
END_VAR
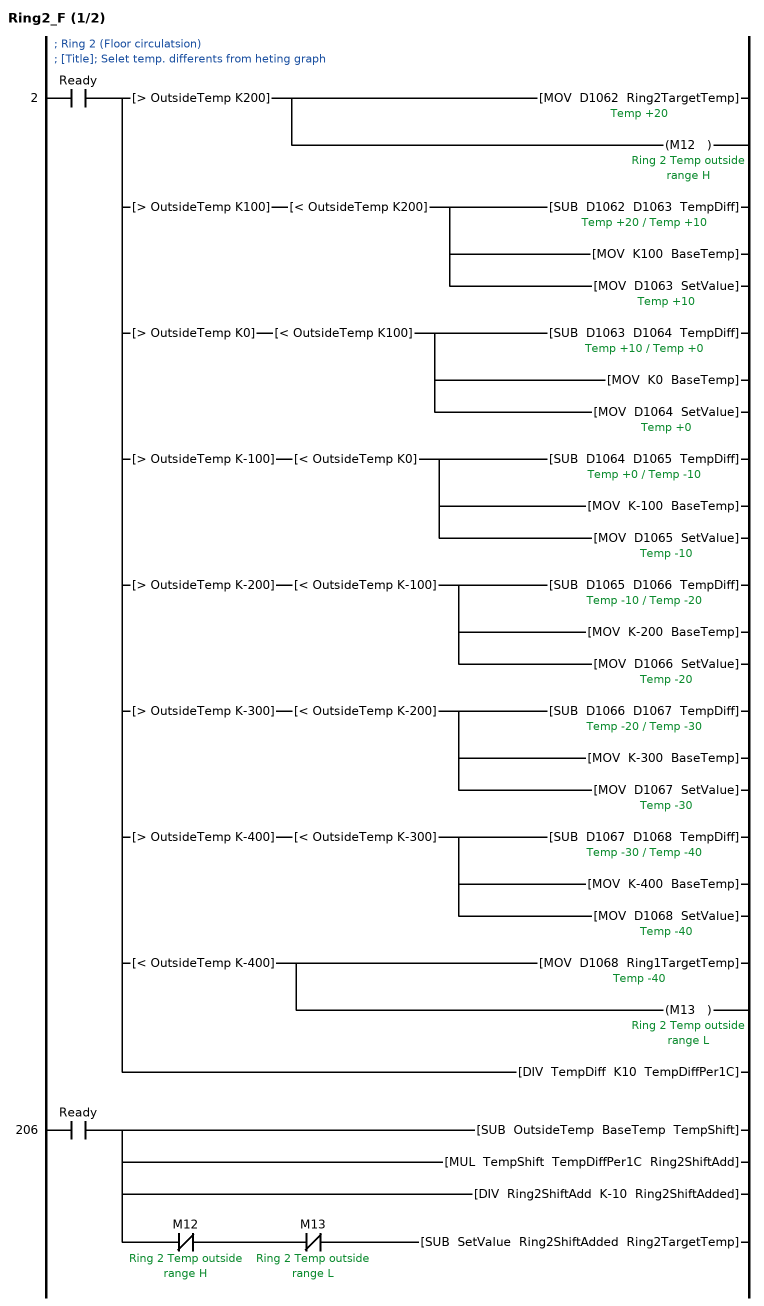
; Ring 2 (Floor circulatsion)
; [Title]; Selet temp. differents from heting graph
2     LD      Ready
      MPS
      AND>    OutsideTemp K200
      MOV     D1062 Ring2TargetTemp  ; Temp +20
        [note] Data from heating graph
      OUT     M12  ; Ring 2 Temp outside range H
      MRD
      AND>    OutsideTemp K100
      AND<    OutsideTemp K200
      SUB     D1062 D1063 TempDiff  ; Temp +10
      MOV     K100 BaseTemp
      MOV     D1063 SetValue
      MRD
      AND>    OutsideTemp K0
      AND<    OutsideTemp K100
      SUB     D1063 D1064 TempDiff  ; Temp +0
      MOV     K0 BaseTemp
      MOV     D1064 SetValue
      MRD
      AND>    OutsideTemp K-100
      AND<    OutsideTemp K0
      SUB     D1064 D1065 TempDiff  ; Temp -10
      MOV     K-100 BaseTemp
      MOV     D1065 SetValue
      MRD
      AND>    OutsideTemp K-200
      AND<    OutsideTemp K-100
      SUB     D1065 D1066 TempDiff  ; Temp -20
      MOV     K-200 BaseTemp
      MOV     D1066 SetValue
      MRD
      AND>    OutsideTemp K-300
      AND<    OutsideTemp K-200
      SUB     D1066 D1067 TempDiff  ; Temp -30
      MOV     K-300 BaseTemp
      MOV     D1067 SetValue
      MRD
      AND>    OutsideTemp K-400
      AND<    OutsideTemp K-300
      SUB     D1067 D1068 TempDiff  ; Temp -40
      MOV     K-400 BaseTemp
      MOV     D1068 SetValue
      MRD
      AND<    OutsideTemp K-400
      MOV     D1068 Ring1TargetTemp
        [note] Data from heating graph
      OUT     M13  ; Ring 2 Temp outside range L
      MPP
      DIV     TempDiff K10 TempDiffPer1C
        [note] Calculated differents per 1C
206   LD      Ready
      SUB     OutsideTemp BaseTemp TempShift
        [note] Temp differents
      MUL     TempShift TempDiffPer1C Ring2ShiftAdd
        [note] Temp diffrents  per 1C
      DIV     Ring2ShiftAdd K-10 Ring2ShiftAdded
      ANI     M12  ; Ring 2 Temp outside range H
      ANI     M13  ; Ring 2 Temp outside range L
      SUB     SetValue Ring2ShiftAdded Ring2TargetTemp
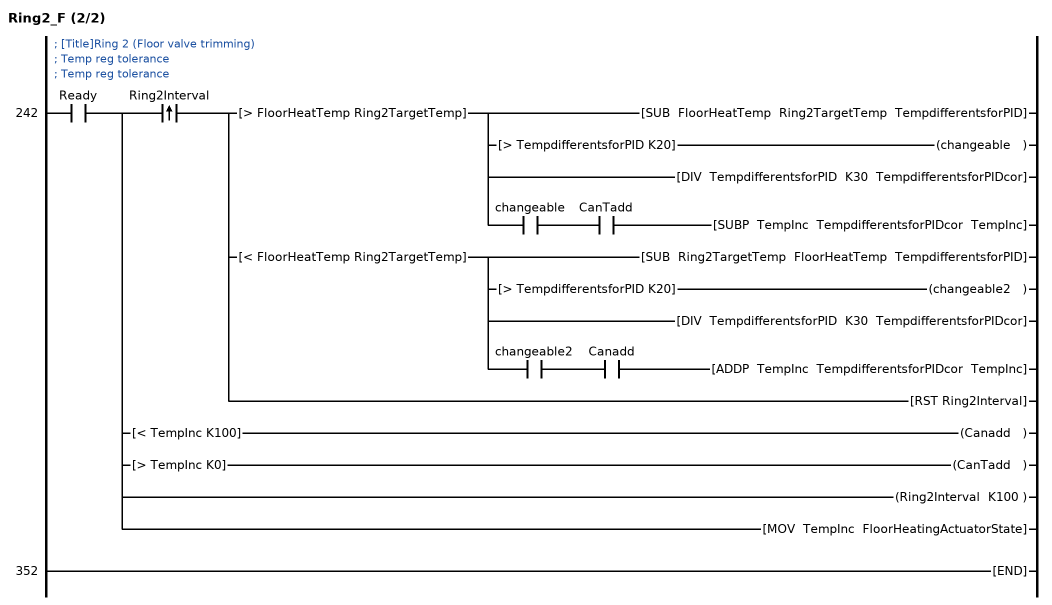
; [Title]Ring 2 (Floor valve trimming)
; Temp reg tolerance
; Temp reg tolerance
242   LD      Ready
      MPS
      ANDP    Ring2Interval
      MPS
      AND>    FloorHeatTemp Ring2TargetTemp
      SUB     FloorHeatTemp Ring2TargetTemp TempdifferentsforPID
        [note] Calc temp differents for PID
      MPS
      AND>    TempdifferentsforPID K20
      OUT     changeable
        [note] Temp reg tolerance
      MPP
      DIV     TempdifferentsforPID K30 TempdifferentsforPIDcor
        [note] PID to actuator (%)
      AND     changeable
      AND     CanTadd
      SUBP    TempInc TempdifferentsforPIDcor TempInc
        [note] Correctsion actuator value (%)
      MRD
      AND<    FloorHeatTemp Ring2TargetTemp
      SUB     Ring2TargetTemp FloorHeatTemp TempdifferentsforPID
        [note] Calc temp differents for PID
      MPS
      AND>    TempdifferentsforPID K20
      OUT     changeable2
        [note] Temp reg tolerance
      MPP
      DIV     TempdifferentsforPID K30 TempdifferentsforPIDcor
        [note] PID to actuator (%)
      AND     changeable2
      AND     Canadd
      ADDP    TempInc TempdifferentsforPIDcor TempInc
        [note] Correctsion actuator value (%)
      MPP
      RST     Ring2Interval
      MRD
      AND<    TempInc K100
      OUT     Canadd
        [note] Actuator range control
      MRD
      AND>    TempInc K0
      OUT     CanTadd
      MPP
      OUT     Ring2Interval K100
      MOV     TempInc FloorHeatingActuatorState
352   END
END_PROGRAM

PROGRAM El_Heat
VAR
  TempDiffPer1C : DINT;  (* Temerature differents pes 1 C *)
  TempShift : DINT;  (* Temperature shift *)
  Ring2ShiftAdd : DINT;
  Ring2ShiftAdded : DINT;
  TempDiff : DINT;  (* Heat Graph temp difference *)
  BaseTemp : INT;  (* Base temperatuere for calc *)
  SetValue : INT;  (* Value from Graph *)
  Ring2Interval : TIMER;  (* Ring 1 actuator valve update interval *)
  TempdifferentsforPID : INT;  (* Temp different for PID *)
  TempInc : INT;  (* Temperature increment to actuator *)
  Ring1Interval : TIMER;  (* Ring 1 actuator valve update interval *)
  changeable : BOOL;  (* temperatuure need correctsion *)
  TempdifferentsforPIDcor : DINT;  (* Corrected actuator value change *)
  Canadd : BOOL;  (* Can add more value *)
  CanTadd : BOOL;  (* Cant add more val *)
  changeable2 : BOOL;
  El_Heat_ON : BOOL;  (* Electric heat func is activ *)
END_VAR
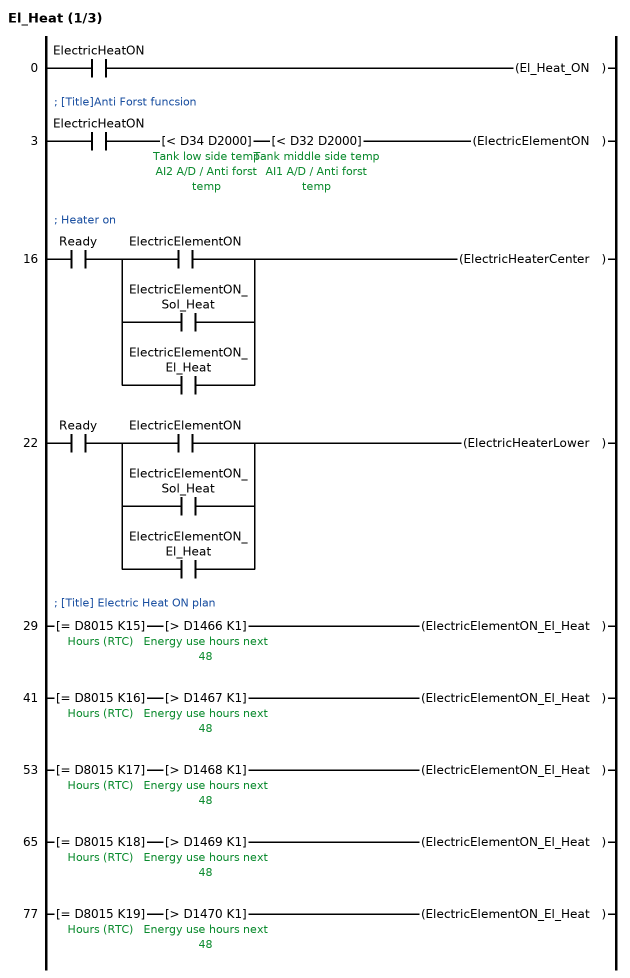
0     LD      ElectricHeatON
      OUT     El_Heat_ON
; [Title]Anti Forst funcsion
3     LD      ElectricHeatON
      AND<    D34 D2000  ; Tank low side temp AI2 A/D / Anti forst temp
      AND<    D32 D2000  ; Tank middle side temp AI1 A/D / Anti forst temp
      OUT     ElectricElementON
; Heater on
16    LD      Ready
      LD      ElectricElementON
      OR      ElectricElementON_Sol_Heat
      OR      ElectricElementON_El_Heat
      ANB
      OUT     ElectricHeaterCenter
22    LD      Ready
      LD      ElectricElementON
      OR      ElectricElementON_Sol_Heat
      OR      ElectricElementON_El_Heat
      ANB
      OUT     ElectricHeaterLower
; [Title] Electric Heat ON plan
29    LD=     D8015 K15  ; Hours (RTC)
      AND>    D1466 K1  ; Energy use hours next 48
      OUT     ElectricElementON_El_Heat
        [note] 15,00
41    LD=     D8015 K16  ; Hours (RTC)
      AND>    D1467 K1  ; Energy use hours next 48
      OUT     ElectricElementON_El_Heat
        [note] 16,00
53    LD=     D8015 K17  ; Hours (RTC)
      AND>    D1468 K1  ; Energy use hours next 48
      OUT     ElectricElementON_El_Heat
        [note] 17,00
65    LD=     D8015 K18  ; Hours (RTC)
      AND>    D1469 K1  ; Energy use hours next 48
      OUT     ElectricElementON_El_Heat
        [note] 18,00
77    LD=     D8015 K19  ; Hours (RTC)
      AND>    D1470 K1  ; Energy use hours next 48
      OUT     ElectricElementON_El_Heat
        [note] 19,00
